SUBAPPLICATION Uebung_017 (* Subapplication Type *)
  (* Standard: 61499-2 *)
  (* Version 1.0, 2023-10-23, franz *)
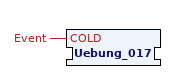
  EVENT_INPUT
    COLD;
  END_EVENT
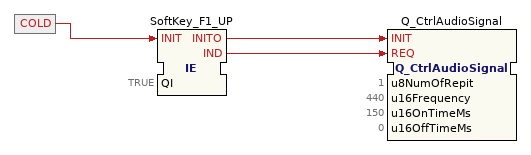
  FBS
    SoftKey_F1_UP : IE(QI := TRUE);
    Q_CtrlAudioSignal : Q_CtrlAudioSignal(u8NumOfRepit := 1, u16Frequency := 440, u16OnTimeMs := 150, u16OffTimeMs := 0);
  END_FBS
  EVENT_CONNECTIONS
    COLD TO SoftKey_F1_UP.INIT;
    SoftKey_F1_UP.INITO TO Q_CtrlAudioSignal.INIT;
    SoftKey_F1_UP.IND TO Q_CtrlAudioSignal.REQ;
  END_CONNECTIONS
END_SUBAPPLICATION
